// TIA Portal project "MB TCP S7-1200 - HMI ET6600" (V19)

(* hardware
DEVICE "S7-1200 station_1"  S7-1200 Station
   slot 0: "Rack_0"  S7-1200 Rack  Rack  V1.0
   slot 1: "PLC_1"  CPU 1215C DC/DC/DC  6ES7 215-1AG40-0XB0  V4.5
*)

// ===== PLC "PLC_1"  CPU 1215C DC/DC/DC =====

VAR_GLOBAL   // PLC tag table "Default tag table"
   "Encendido" AT %M0.0 : Bool;
   "ManAuto" AT %M0.1 : Bool;
   "System_Byte" AT %MB1 : Byte;
   "FirstScan" AT %M1.0 : Bool;
   "DiagStatusUpdate" AT %M1.1 : Bool;
   "AlwaysTRUE" AT %M1.2 : Bool;
   "AlwaysFALSE" AT %M1.3 : Bool;
END_VAR

DATA_BLOCK "DB_AproxTemp"   // DB1
{ S7_Optimized_Access := 'TRUE' }
VERSION : 0.1
// stored: InstanceOfName FB_Aprox
"FB_Aprox"
BEGIN
END_DATA_BLOCK

DATA_BLOCK "DB_HMIET"   // DB2
{ S7_Optimized_Access := 'FALSE' }
VERSION : 0.1
   VAR
      TEMPERATURA_SP : Real := 22.0;
      HUMEDAD_SP : Real := 60.0;
      PRESION_SP : Real := 1015.0;
      VENT_VEL_OUT : Real := 799.0;
      BOMBA_VEL_OUT : Real := 1434.0;
      TEMPERATURA_HMI : Int;
      HUMEDAD_HMI : Int;
      PRESION_HMI : Int;
      ENFRIAMIENTO_HMI : Bool;
      CALEFACCION_HMI : Bool;
      DESHUM_HMI : Bool;
      AutoMan : Bool;
      CAUDAL_BS : Int;
      MrgPre : Real;
   END_VAR
BEGIN
END_DATA_BLOCK

DATA_BLOCK "DB_AproxHum"   // DB3
{ S7_Optimized_Access := 'TRUE' }
VERSION : 0.1
// stored: InstanceOfName FB_Aprox
"FB_Aprox"
BEGIN
END_DATA_BLOCK

DATA_BLOCK "DB_AproxPre"   // DB4
{ S7_Optimized_Access := 'TRUE' }
VERSION : 0.1
// stored: InstanceOfName FB_Aprox
"FB_Aprox"
BEGIN
END_DATA_BLOCK

DATA_BLOCK "DB_SimTemp"   // DB5
{ S7_Optimized_Access := 'TRUE' }
VERSION : 0.1
// stored: InstanceOfName FB_Simulacion
"FB_Simulacion"
BEGIN
END_DATA_BLOCK

DATA_BLOCK "DB_SimPre"   // DB6
{ S7_Optimized_Access := 'TRUE' }
VERSION : 0.1
// stored: InstanceOfName FB_Simulacion
"FB_Simulacion"
BEGIN
END_DATA_BLOCK

DATA_BLOCK "DB_HMIOUT"   // DB7
{ S7_Optimized_Access := 'FALSE' }
VERSION : 0.1
   VAR
      PRESION_OUT : Real;
      HUMEDAD_OUT : Real;
      TEMPERATURA_OUT : Real;
      TENSION_OUT : Real;
      CORRIENTE_OUT : Real;
      VELOCIDAD_OUT : Real;
      PPM_PRC : Int;
      PPM_OUT : Int;
      ALARMA_BS : Bool;
   END_VAR
BEGIN
END_DATA_BLOCK

DATA_BLOCK "DB_OsciladorTension"   // DB8
{ S7_Optimized_Access := 'TRUE' }
VERSION : 0.1
// stored: InstanceOfName FB_Oscilador
"FB_Oscilador"
BEGIN
END_DATA_BLOCK

DATA_BLOCK "DB_OsciladorCorriente"   // DB9
{ S7_Optimized_Access := 'TRUE' }
VERSION : 0.1
// stored: InstanceOfName FB_Oscilador
"FB_Oscilador"
BEGIN
END_DATA_BLOCK

DATA_BLOCK "DB_OsciladorVel"   // DB10
{ S7_Optimized_Access := 'TRUE' }
VERSION : 0.1
// stored: InstanceOfName FB_Oscilador
"FB_Oscilador"
BEGIN
END_DATA_BLOCK

DATA_BLOCK "DB_CaliAire"   // DB11
{ S7_Optimized_Access := 'TRUE' }
VERSION : 0.1
// stored: InstanceOfName FB_CaliAire
"FB_CaliAire"
BEGIN
END_DATA_BLOCK

DATA_BLOCK "DB_SimHum"   // DB12
{ S7_Optimized_Access := 'TRUE' }
VERSION : 0.1
// stored: InstanceOfName FB_Simulacion
"FB_Simulacion"
BEGIN
END_DATA_BLOCK

// folder: System blocks/Program resources

DATA_BLOCK "Timer_VelBombaVent"   // DB13
{ S7_Optimized_Access := 'TRUE' }
AUTHOR : Simatic
FAMILY : IEC
NAME : IEC_TMR
VERSION : 1.0
// stored: InstanceOfName IEC_TIMER
"IEC_TIMER"
BEGIN
END_DATA_BLOCK

// folder: (top level)

FUNCTION_BLOCK "FB_Oscilador"   // FB1, LAD
{ S7_Optimized_Access := 'TRUE' }
VERSION : 0.1
   VAR_INPUT
      SP : Real;
      MS : Real;
      MI : Real;
      Tiempo : Time;
      Enc : Bool;
   END_VAR
   VAR_OUTPUT
      PV : Real;
   END_VAR
   VAR
      Timer_MS : TON_TIME;
      Reset_TMS : Bool;
      Timer_ResetMS : TON_TIME;
      Intermedio : Bool;
      Reset_TMI : Bool;
      Timer_MI : TON_TIME;
      Timer_ResetMI : TON_TIME;
   END_VAR
BEGIN

REGION Network 1
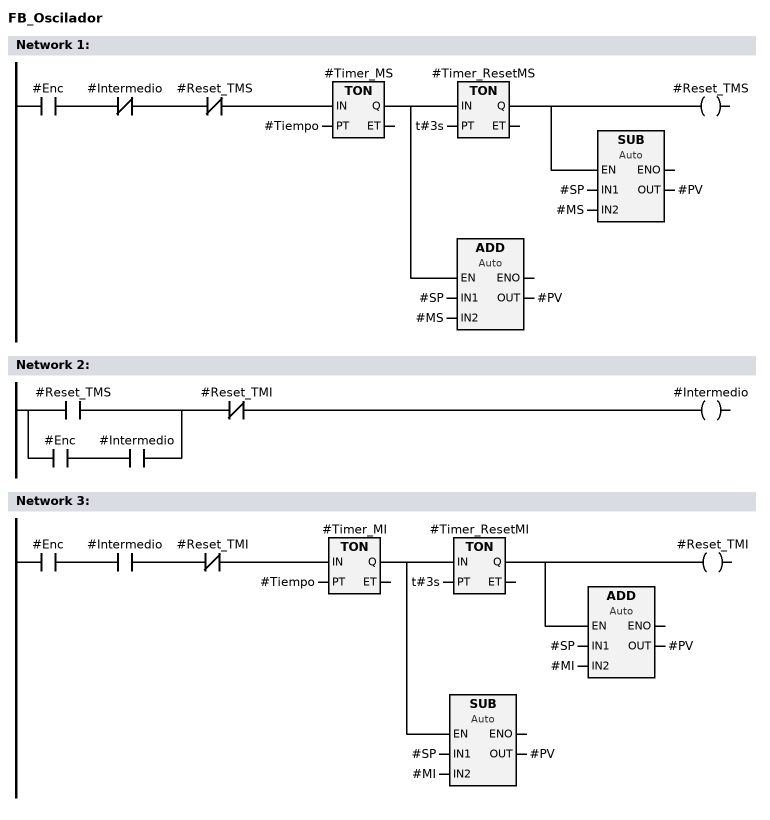
   #Timer_MS(IN := #Enc AND NOT #Intermedio AND NOT #Reset_TMS, PT := #Tiempo);   // TON
   #Timer_ResetMS(IN := #Timer_MS.Q, PT := t#3s);   // TON
   #Reset_TMS := #Timer_ResetMS.Q;
   IF #Timer_ResetMS.Q THEN #PV := #SP - #MS; END_IF;
   IF #Timer_MS.Q THEN #PV := #SP + #MS; END_IF;
END_REGION

REGION Network 2
   RUNG wire#powerrail
      Contact( #Reset_TMS )
      wire#w1
      I_Contact( #Reset_TMI )
      Coil( #Intermedio )
   END_RUNG
   RUNG wire#powerrail
      Contact( #Enc )
      Contact( #Intermedio )
   END_RUNG wire#w1
   // the same network as SCL:
   #Intermedio := (#Reset_TMS OR (#Enc AND #Intermedio)) AND NOT #Reset_TMI;
END_REGION

REGION Network 3
   #Timer_MI(IN := #Enc AND #Intermedio AND NOT #Reset_TMI, PT := #Tiempo);   // TON
   #Timer_ResetMI(IN := #Timer_MI.Q, PT := t#3s);   // TON
   #Reset_TMI := #Timer_ResetMI.Q;
   IF #Timer_ResetMI.Q THEN #PV := #SP + #MI; END_IF;
   IF #Timer_MI.Q THEN #PV := #SP - #MI; END_IF;
END_REGION
END_FUNCTION_BLOCK

FUNCTION_BLOCK "FB_Simulacion"   // FB2, LAD
{ S7_Optimized_Access := 'TRUE' }
VERSION : 0.1
   VAR_INPUT
      Enc : Bool;
      Mrg : Real;
   END_VAR
   VAR_OUTPUT
      PV : Real;
      Ctrl : Int;
      Sim : Bool;
   END_VAR
   VAR
      Aux : Array[0..7] of Bool;
      MarcaEnc : Bool;
      TimerSuma : TON_TIME;
      TimerEnclavSuma : TON_TIME;
      TimerDelay : TON_TIME;
      TimerEnclavResta : TON_TIME;
   END_VAR
   VAR_TEMP   // added for the SCL form of the ladder/FBD networks
      _w1 : Bool;
   END_VAR
BEGIN

REGION Network 1
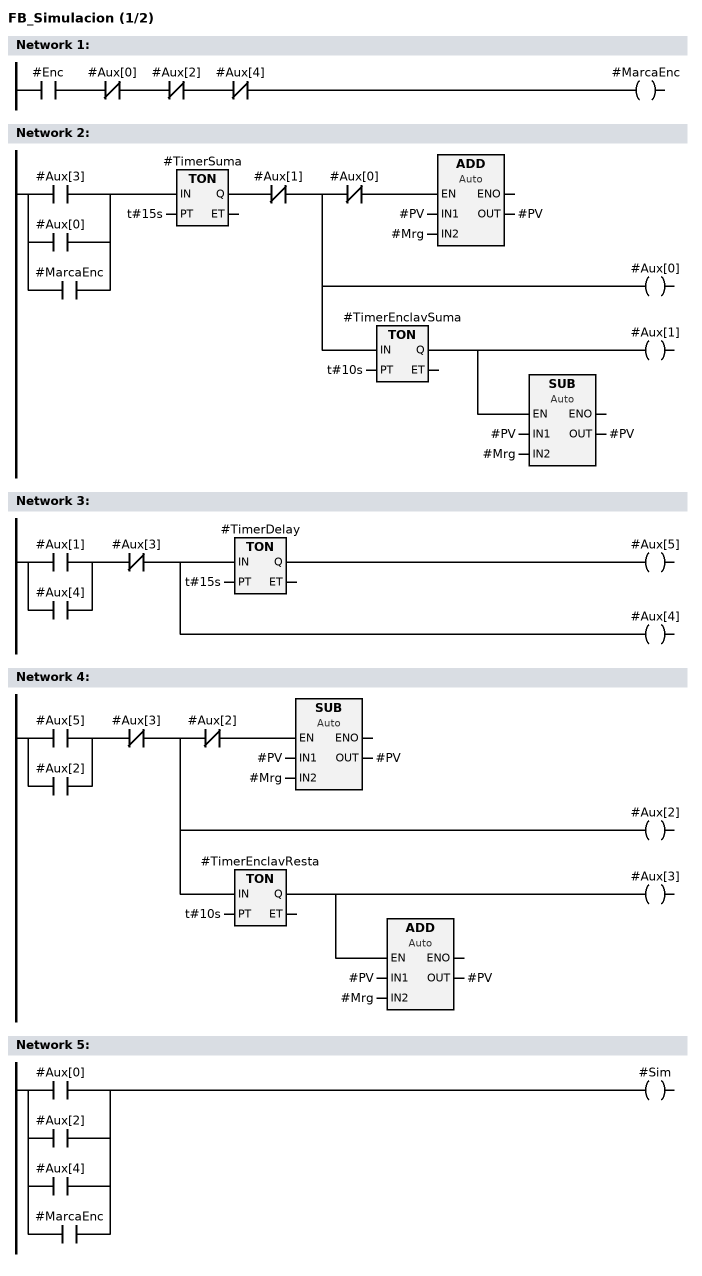
   RUNG wire#powerrail
      Contact( #Enc )
      I_Contact( #Aux[0] )
      I_Contact( #Aux[2] )
      I_Contact( #Aux[4] )
      Coil( #MarcaEnc )
   END_RUNG
   // the same network as SCL:
   #MarcaEnc := #Enc AND NOT #Aux[0] AND NOT #Aux[2] AND NOT #Aux[4];
END_REGION

REGION Network 2
   #TimerSuma(IN := #Aux[3] OR #Aux[0] OR #MarcaEnc, PT := t#15s);   // TON
   #_w1 := #TimerSuma.Q AND NOT #Aux[1];
   IF #_w1 AND NOT #Aux[0] THEN #PV := #PV + #Mrg; END_IF;
   #Aux[0] := #_w1;
   #TimerEnclavSuma(IN := #_w1, PT := t#10s);   // TON
   #Aux[1] := #TimerEnclavSuma.Q;
   IF #TimerEnclavSuma.Q THEN #PV := #PV - #Mrg; END_IF;
END_REGION

REGION Network 3
   #_w1 := (#Aux[1] OR #Aux[4]) AND NOT #Aux[3];
   #TimerDelay(IN := #_w1, PT := t#15s);   // TON
   #Aux[5] := #TimerDelay.Q;
   #Aux[4] := #_w1;
END_REGION

REGION Network 4
   #_w1 := (#Aux[5] OR #Aux[2]) AND NOT #Aux[3];
   IF #_w1 AND NOT #Aux[2] THEN #PV := #PV - #Mrg; END_IF;
   #Aux[2] := #_w1;
   #TimerEnclavResta(IN := #_w1, PT := t#10s);   // TON
   #Aux[3] := #TimerEnclavResta.Q;
   IF #TimerEnclavResta.Q THEN #PV := #PV + #Mrg; END_IF;
END_REGION

REGION Network 5
   RUNG wire#powerrail
      Contact( #Aux[0] )
      wire#w1
      Coil( #Sim )
   END_RUNG
   RUNG wire#powerrail
      Contact( #Aux[2] )
   END_RUNG wire#w1
   RUNG wire#powerrail
      Contact( #Aux[4] )
   END_RUNG wire#w1
   RUNG wire#powerrail
      Contact( #MarcaEnc )
   END_RUNG wire#w1
   // the same network as SCL:
   #Sim := #Aux[0] OR #Aux[2] OR #Aux[4] OR #MarcaEnc;
END_REGION

REGION Network 6
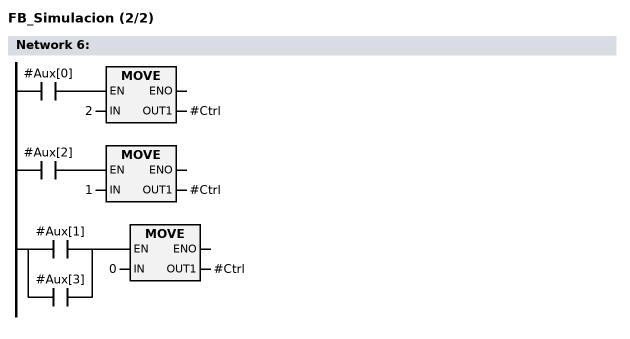
   RUNG wire#powerrail
      Contact( #Aux[0] )
      Move(in := 2, out1 => #Ctrl)
   END_RUNG
   RUNG wire#powerrail
      Contact( #Aux[2] )
      Move(in := 1, out1 => #Ctrl)
   END_RUNG
   RUNG wire#powerrail
      Contact( #Aux[1] )
      wire#w1
      Move(in := 0, out1 => #Ctrl)
   END_RUNG
   RUNG wire#powerrail
      Contact( #Aux[3] )
   END_RUNG wire#w1
   // the same network as SCL:
   IF #Aux[0] THEN #Ctrl := 2; END_IF;
   IF #Aux[2] THEN #Ctrl := 1; END_IF;
   IF #Aux[1] OR #Aux[3] THEN #Ctrl := 0; END_IF;
END_REGION
END_FUNCTION_BLOCK

FUNCTION_BLOCK "FB_CaliAire"   // FB3, LAD
{ S7_Optimized_Access := 'TRUE' }
VERSION : 0.1
   VAR_INPUT
      Caudal : Int;
      Lim : Int;
   END_VAR
   VAR_OUTPUT
      PPM : Int;
      PPMEsc : Int;
      Alarma : Bool;
   END_VAR
   VAR
      UltCaudal : Int := 100;
      TempOn : Bool;
      Timer_CaliAire : TON_TIME;
      TempPPM : Real;
   END_VAR
BEGIN

REGION Network 1
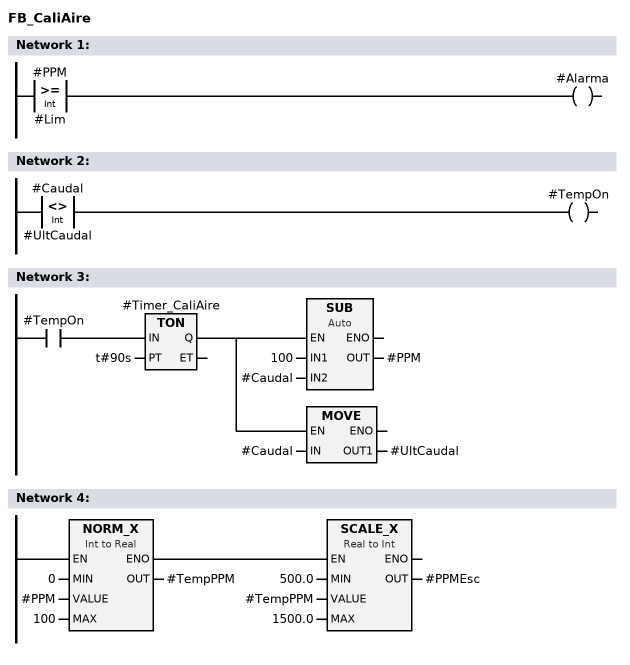
   RUNG wire#powerrail
      { S7_Templates := "SrcType := Int" } GE_Contact(in1 := #PPM, in2 := #Lim)
      Coil( #Alarma )
   END_RUNG
   // the same network as SCL:
   #Alarma := #PPM >= #Lim;
END_REGION

REGION Network 2
   RUNG wire#powerrail
      { S7_Templates := "SrcType := Int" } NE_Contact(in1 := #Caudal, in2 := #UltCaudal)
      Coil( #TempOn )
   END_RUNG
   // the same network as SCL:
   #TempOn := #Caudal <> #UltCaudal;
END_REGION

REGION Network 3
   #Timer_CaliAire(IN := #TempOn, PT := t#90s);   // TON
   IF #Timer_CaliAire.Q THEN
       #PPM := 100 - #Caudal;
       #UltCaudal := #Caudal;
   END_IF;
END_REGION

REGION Network 4
   RUNG wire#powerrail
      { S7_Templates := "[SrcType := Int, DestType := Real]" } Normalize(min := 0, value := #PPM, max := 100, out => #TempPPM)
      { S7_Templates := "[SrcType := Real, DestType := Int]" } Scale(min := 500.0, value := #TempPPM, max := 1500.0, out => #PPMEsc)
   END_RUNG
   // the same network as SCL:
   #TempPPM := NORM_X(MIN := 0, VALUE := #PPM, MAX := 100);
   #PPMEsc := SCALE_X(MIN := 500.0, VALUE := #TempPPM, MAX := 1500.0);
END_REGION
END_FUNCTION_BLOCK

FUNCTION_BLOCK "FB_Aprox"   // FB4, LAD
{ S7_Optimized_Access := 'TRUE' }
VERSION : 0.1
   VAR_INPUT
      Enc : Bool;
      SP : Real;
      Mrg : Real;
   END_VAR
   VAR_OUTPUT
      PV : Real;
      Ctrl : Int;
   END_VAR
   VAR
      Aux : Array[0..7] of Bool;
      TimerAprox : TON_TIME;
   END_VAR
BEGIN

REGION Network 1
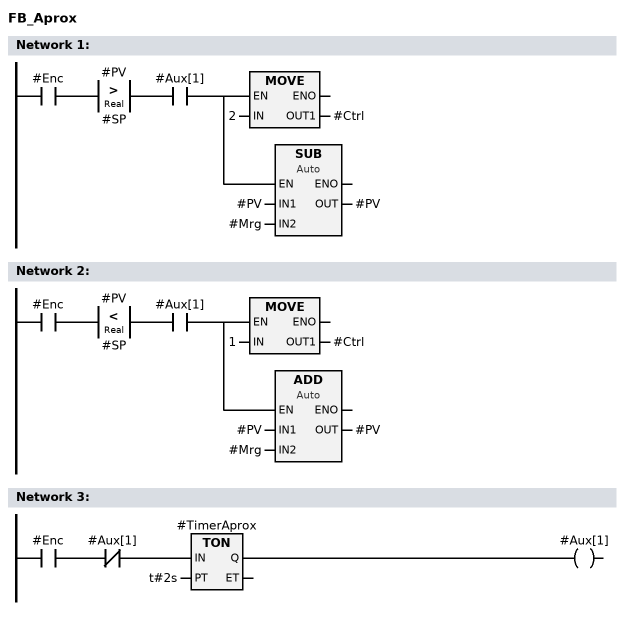
   RUNG wire#powerrail
      Contact( #Enc )
      { S7_Templates := "SrcType := Real" } GT_Contact(in1 := #PV, in2 := #SP)
      Contact( #Aux[1] )
      wire#w1
      Move(in := 2, out1 => #Ctrl)
   END_RUNG
   RUNG wire#w1
      Sub(in1 := #PV, in2 := #Mrg, out => #PV)
   END_RUNG
   // the same network as SCL:
   IF #Enc AND (#PV > #SP) AND #Aux[1] THEN
       #Ctrl := 2;
       #PV := #PV - #Mrg;
   END_IF;
END_REGION

REGION Network 2
   RUNG wire#powerrail
      Contact( #Enc )
      { S7_Templates := "SrcType := Real" } LT_Contact(in1 := #PV, in2 := #SP)
      Contact( #Aux[1] )
      wire#w1
      Move(in := 1, out1 => #Ctrl)
   END_RUNG
   RUNG wire#w1
      Add(in1 := #PV, in2 := #Mrg, out => #PV)
   END_RUNG
   // the same network as SCL:
   IF #Enc AND (#PV < #SP) AND #Aux[1] THEN
       #Ctrl := 1;
       #PV := #PV + #Mrg;
   END_IF;
END_REGION

REGION Network 3
   #TimerAprox(IN := #Enc AND NOT #Aux[1], PT := t#2s);   // TON
   #Aux[1] := #TimerAprox.Q;
END_REGION
END_FUNCTION_BLOCK

FUNCTION_BLOCK "Modbus_TCP"   // FB5, LAD
{ S7_Optimized_Access := 'TRUE' }
VERSION : 0.1
BEGIN
END_FUNCTION_BLOCK

FUNCTION "FC_ConversionEscalado" : Void   // FC1, LAD
{ S7_Optimized_Access := 'TRUE' }
VERSION : 0.1
   VAR_INPUT
      EntradaInt : Int;
      MinNorm : Int;
      MaxNorm : Int;
      MinReal : Real;
      MaxReal : Real;
   END_VAR
   VAR_OUTPUT
      SalidaReal : Real;
   END_VAR
   VAR_TEMP
      IntReal : Real;
      RealNorm : Real;
   END_VAR
BEGIN

REGION Network 1
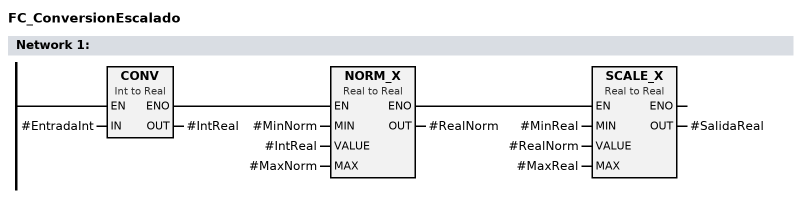
   RUNG wire#powerrail
      { S7_Templates := "[SrcType := Int, DestType := Real]" } Convert(in := #EntradaInt, out => #IntReal)
      { S7_Templates := "[SrcType := Real, DestType := Real]" } Normalize(min := #MinNorm, value := #IntReal, max := #MaxNorm, out => #RealNorm)
      { S7_Templates := "[SrcType := Real, DestType := Real]" } Scale(min := #MinReal, value := #RealNorm, max := #MaxReal, out => #SalidaReal)
   END_RUNG
   // the same network as SCL:
   #IntReal := INT_TO_REAL(#EntradaInt);
   #RealNorm := NORM_X(MIN := #MinNorm, VALUE := #IntReal, MAX := #MaxNorm);
   #SalidaReal := SCALE_X(MIN := #MinReal, VALUE := #RealNorm, MAX := #MaxReal);
END_REGION
END_FUNCTION

ORGANIZATION_BLOCK "Main"   // OB1, LAD, ProgramCycle
TITLE = "Main Program Sweep (Cycle)"
{ S7_Optimized_Access := 'TRUE' }
VERSION : 0.1
   VAR_INPUT
      Initial_Call : Bool;   // Initial call of this OB
      Remanence : Bool;   // =True, if remanent data are available
   END_VAR
   VAR_TEMP
      SPTEMP_ESC : Real;
      SPHUM_ESC : Real;
      SPPRE_ESC : Real;
   END_VAR
BEGIN

REGION Network 1
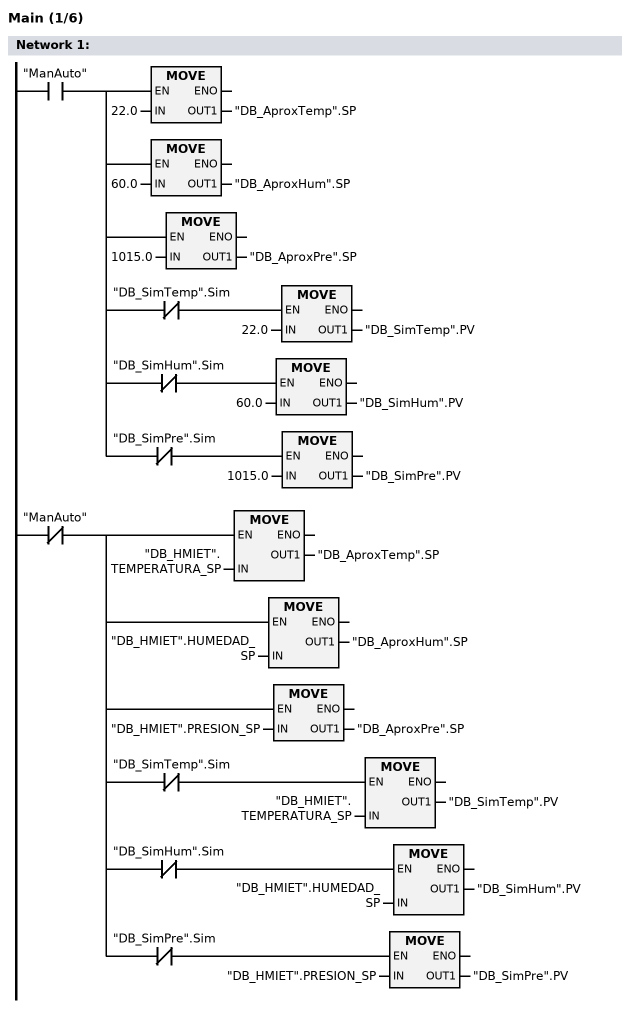
   RUNG wire#powerrail
      Contact( "ManAuto" )
      wire#w1
      Move(in := 22.0, out1 => "DB_AproxTemp".SP)
   END_RUNG
   RUNG wire#w1
      Move(in := 60.0, out1 => "DB_AproxHum".SP)
   END_RUNG
   RUNG wire#w1
      Move(in := 1015.0, out1 => "DB_AproxPre".SP)
   END_RUNG
   RUNG wire#w1
      I_Contact( "DB_SimTemp".Sim )
      Move(in := 22.0, out1 => "DB_SimTemp".PV)
   END_RUNG
   RUNG wire#w1
      I_Contact( "DB_SimHum".Sim )
      Move(in := 60.0, out1 => "DB_SimHum".PV)
   END_RUNG
   RUNG wire#w1
      I_Contact( "DB_SimPre".Sim )
      Move(in := 1015.0, out1 => "DB_SimPre".PV)
   END_RUNG
   RUNG wire#powerrail
      I_Contact( "ManAuto" )
      wire#w2
      Move(in := "DB_HMIET".TEMPERATURA_SP, out1 => "DB_AproxTemp".SP)
   END_RUNG
   RUNG wire#w2
      Move(in := "DB_HMIET".HUMEDAD_SP, out1 => "DB_AproxHum".SP)
   END_RUNG
   RUNG wire#w2
      Move(in := "DB_HMIET".PRESION_SP, out1 => "DB_AproxPre".SP)
   END_RUNG
   RUNG wire#w2
      I_Contact( "DB_SimTemp".Sim )
      Move(in := "DB_HMIET".TEMPERATURA_SP, out1 => "DB_SimTemp".PV)
   END_RUNG
   RUNG wire#w2
      I_Contact( "DB_SimHum".Sim )
      Move(in := "DB_HMIET".HUMEDAD_SP, out1 => "DB_SimHum".PV)
   END_RUNG
   RUNG wire#w2
      I_Contact( "DB_SimPre".Sim )
      Move(in := "DB_HMIET".PRESION_SP, out1 => "DB_SimPre".PV)
   END_RUNG
   // the same network as SCL:
   IF "ManAuto" THEN
       "DB_AproxTemp".SP := 22.0;
       "DB_AproxHum".SP := 60.0;
       "DB_AproxPre".SP := 1015.0;
   END_IF;
   IF "ManAuto" AND NOT "DB_SimTemp".Sim THEN "DB_SimTemp".PV := 22.0; END_IF;
   IF "ManAuto" AND NOT "DB_SimHum".Sim THEN "DB_SimHum".PV := 60.0; END_IF;
   IF "ManAuto" AND NOT "DB_SimPre".Sim THEN "DB_SimPre".PV := 1015.0; END_IF;
   IF NOT "ManAuto" THEN
       "DB_AproxTemp".SP := "DB_HMIET".TEMPERATURA_SP;
       "DB_AproxHum".SP := "DB_HMIET".HUMEDAD_SP;
       "DB_AproxPre".SP := "DB_HMIET".PRESION_SP;
   END_IF;
   IF NOT "ManAuto" AND NOT "DB_SimTemp".Sim THEN "DB_SimTemp".PV := "DB_HMIET".TEMPERATURA_SP; END_IF;
   IF NOT "ManAuto" AND NOT "DB_SimHum".Sim THEN "DB_SimHum".PV := "DB_HMIET".HUMEDAD_SP; END_IF;
   IF NOT "ManAuto" AND NOT "DB_SimPre".Sim THEN "DB_SimPre".PV := "DB_HMIET".PRESION_SP; END_IF;
END_REGION

REGION Network 2
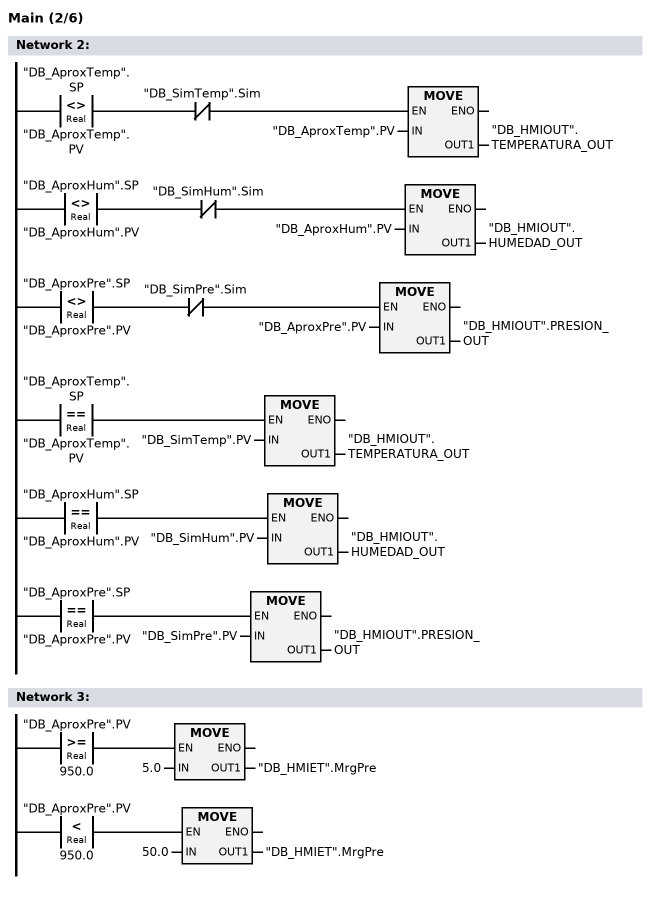
   RUNG wire#powerrail
      { S7_Templates := "SrcType := Real" } NE_Contact(in1 := "DB_AproxTemp".SP, in2 := "DB_AproxTemp".PV)
      I_Contact( "DB_SimTemp".Sim )
      Move(in := "DB_AproxTemp".PV, out1 => "DB_HMIOUT".TEMPERATURA_OUT)
   END_RUNG
   RUNG wire#powerrail
      { S7_Templates := "SrcType := Real" } NE_Contact(in1 := "DB_AproxHum".SP, in2 := "DB_AproxHum".PV)
      I_Contact( "DB_SimHum".Sim )
      Move(in := "DB_AproxHum".PV, out1 => "DB_HMIOUT".HUMEDAD_OUT)
   END_RUNG
   RUNG wire#powerrail
      { S7_Templates := "SrcType := Real" } NE_Contact(in1 := "DB_AproxPre".SP, in2 := "DB_AproxPre".PV)
      I_Contact( "DB_SimPre".Sim )
      Move(in := "DB_AproxPre".PV, out1 => "DB_HMIOUT".PRESION_OUT)
   END_RUNG
   RUNG wire#powerrail
      { S7_Templates := "SrcType := Real" } EQ_Contact(in1 := "DB_AproxTemp".SP, in2 := "DB_AproxTemp".PV)
      Move(in := "DB_SimTemp".PV, out1 => "DB_HMIOUT".TEMPERATURA_OUT)
   END_RUNG
   RUNG wire#powerrail
      { S7_Templates := "SrcType := Real" } EQ_Contact(in1 := "DB_AproxHum".SP, in2 := "DB_AproxHum".PV)
      Move(in := "DB_SimHum".PV, out1 => "DB_HMIOUT".HUMEDAD_OUT)
   END_RUNG
   RUNG wire#powerrail
      { S7_Templates := "SrcType := Real" } EQ_Contact(in1 := "DB_AproxPre".SP, in2 := "DB_AproxPre".PV)
      Move(in := "DB_SimPre".PV, out1 => "DB_HMIOUT".PRESION_OUT)
   END_RUNG
   // the same network as SCL:
   IF ("DB_AproxTemp".SP <> "DB_AproxTemp".PV) AND NOT "DB_SimTemp".Sim THEN
       "DB_HMIOUT".TEMPERATURA_OUT := "DB_AproxTemp".PV;
   END_IF;
   IF ("DB_AproxHum".SP <> "DB_AproxHum".PV) AND NOT "DB_SimHum".Sim THEN
       "DB_HMIOUT".HUMEDAD_OUT := "DB_AproxHum".PV;
   END_IF;
   IF ("DB_AproxPre".SP <> "DB_AproxPre".PV) AND NOT "DB_SimPre".Sim THEN
       "DB_HMIOUT".PRESION_OUT := "DB_AproxPre".PV;
   END_IF;
   IF "DB_AproxTemp".SP = "DB_AproxTemp".PV THEN "DB_HMIOUT".TEMPERATURA_OUT := "DB_SimTemp".PV; END_IF;
   IF "DB_AproxHum".SP = "DB_AproxHum".PV THEN "DB_HMIOUT".HUMEDAD_OUT := "DB_SimHum".PV; END_IF;
   IF "DB_AproxPre".SP = "DB_AproxPre".PV THEN "DB_HMIOUT".PRESION_OUT := "DB_SimPre".PV; END_IF;
END_REGION

REGION Network 3
   RUNG wire#powerrail
      { S7_Templates := "SrcType := Real" } GE_Contact(in1 := "DB_AproxPre".PV, in2 := 950.0)
      Move(in := 5.0, out1 => "DB_HMIET".MrgPre)
   END_RUNG
   RUNG wire#powerrail
      { S7_Templates := "SrcType := Real" } LT_Contact(in1 := "DB_AproxPre".PV, in2 := 950.0)
      Move(in := 50.0, out1 => "DB_HMIET".MrgPre)
   END_RUNG
   // the same network as SCL:
   IF "DB_AproxPre".PV >= 950.0 THEN "DB_HMIET".MrgPre := 5.0; END_IF;
   IF "DB_AproxPre".PV < 950.0 THEN "DB_HMIET".MrgPre := 50.0; END_IF;
END_REGION

REGION Network 4
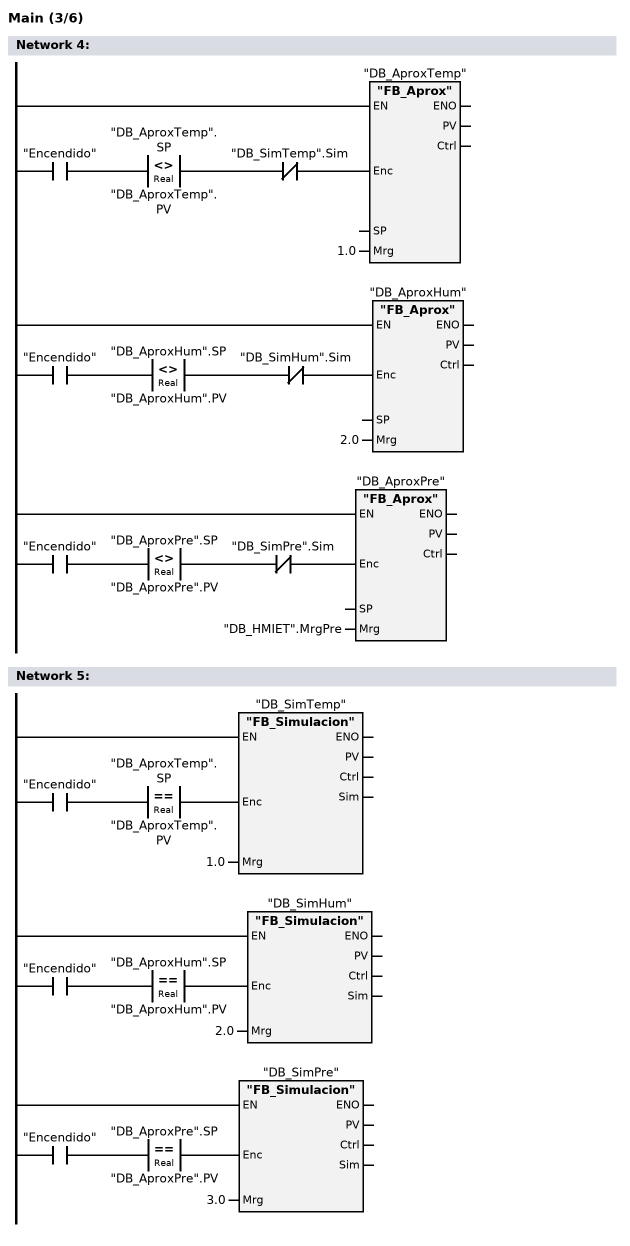
   RUNG wire#powerrail
      "DB_AproxTemp"(Enc := wire#w1, SP :=, Mrg := 1.0, PV =>, Ctrl =>)
   END_RUNG
   RUNG wire#powerrail
      Contact( "Encendido" )
      { S7_Templates := "SrcType := Real" } NE_Contact(in1 := "DB_AproxTemp".SP, in2 := "DB_AproxTemp".PV)
      I_Contact( "DB_SimTemp".Sim )
   END_RUNG wire#w1
   RUNG wire#powerrail
      "DB_AproxHum"(Enc := wire#w2, SP :=, Mrg := 2.0, PV =>, Ctrl =>)
   END_RUNG
   RUNG wire#powerrail
      Contact( "Encendido" )
      { S7_Templates := "SrcType := Real" } NE_Contact(in1 := "DB_AproxHum".SP, in2 := "DB_AproxHum".PV)
      I_Contact( "DB_SimHum".Sim )
   END_RUNG wire#w2
   RUNG wire#powerrail
      "DB_AproxPre"(Enc := wire#w3, SP :=, Mrg := "DB_HMIET".MrgPre, PV =>, Ctrl =>)
   END_RUNG
   RUNG wire#powerrail
      Contact( "Encendido" )
      { S7_Templates := "SrcType := Real" } NE_Contact(in1 := "DB_AproxPre".SP, in2 := "DB_AproxPre".PV)
      I_Contact( "DB_SimPre".Sim )
   END_RUNG wire#w3
   // the same network as SCL:
   "DB_AproxTemp"(Enc := "Encendido" AND ("DB_AproxTemp".SP <> "DB_AproxTemp".PV) AND NOT "DB_SimTemp".Sim,   // "FB_Aprox"
                  Mrg := 1.0);
   "DB_AproxHum"(Enc := "Encendido" AND ("DB_AproxHum".SP <> "DB_AproxHum".PV) AND NOT "DB_SimHum".Sim,   // "FB_Aprox"
                 Mrg := 2.0);
   "DB_AproxPre"(Enc := "Encendido" AND ("DB_AproxPre".SP <> "DB_AproxPre".PV) AND NOT "DB_SimPre".Sim,   // "FB_Aprox"
                 Mrg := "DB_HMIET".MrgPre);
END_REGION

REGION Network 5
   RUNG wire#powerrail
      "DB_SimTemp"(Enc := wire#w1, Mrg := 1.0, PV =>, Ctrl =>, Sim =>)
   END_RUNG
   RUNG wire#powerrail
      Contact( "Encendido" )
      { S7_Templates := "SrcType := Real" } EQ_Contact(in1 := "DB_AproxTemp".SP, in2 := "DB_AproxTemp".PV)
   END_RUNG wire#w1
   RUNG wire#powerrail
      "DB_SimHum"(Enc := wire#w2, Mrg := 2.0, PV =>, Ctrl =>, Sim =>)
   END_RUNG
   RUNG wire#powerrail
      Contact( "Encendido" )
      { S7_Templates := "SrcType := Real" } EQ_Contact(in1 := "DB_AproxHum".SP, in2 := "DB_AproxHum".PV)
   END_RUNG wire#w2
   RUNG wire#powerrail
      "DB_SimPre"(Enc := wire#w3, Mrg := 3.0, PV =>, Ctrl =>, Sim =>)
   END_RUNG
   RUNG wire#powerrail
      Contact( "Encendido" )
      { S7_Templates := "SrcType := Real" } EQ_Contact(in1 := "DB_AproxPre".SP, in2 := "DB_AproxPre".PV)
   END_RUNG wire#w3
   // the same network as SCL:
   "DB_SimTemp"(Enc := "Encendido" AND ("DB_AproxTemp".SP = "DB_AproxTemp".PV), Mrg := 1.0);   // "FB_Simulacion"
   "DB_SimHum"(Enc := "Encendido" AND ("DB_AproxHum".SP = "DB_AproxHum".PV), Mrg := 2.0);   // "FB_Simulacion"
   "DB_SimPre"(Enc := "Encendido" AND ("DB_AproxPre".SP = "DB_AproxPre".PV), Mrg := 3.0);   // "FB_Simulacion"
END_REGION

REGION Network 6
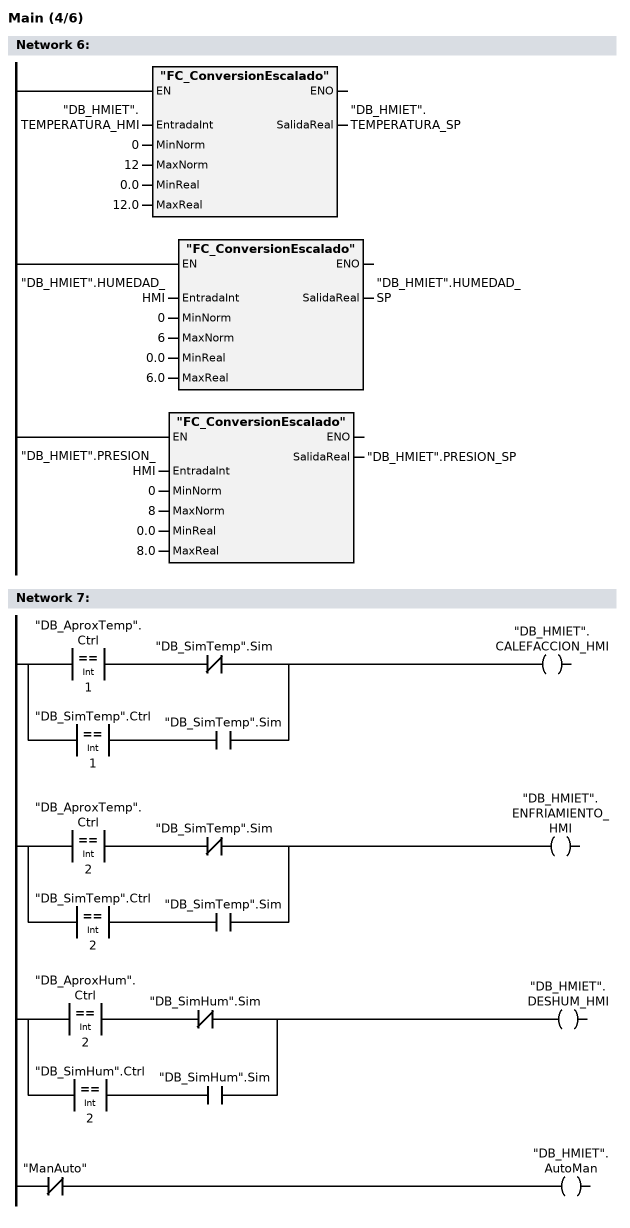
   RUNG wire#powerrail
      "FC_ConversionEscalado"(EntradaInt := "DB_HMIET".TEMPERATURA_HMI, MinNorm := 0, MaxNorm := 12, MinReal := 0.0, MaxReal := 12.0, SalidaReal => "DB_HMIET".TEMPERATURA_SP)
   END_RUNG
   RUNG wire#powerrail
      "FC_ConversionEscalado"(EntradaInt := "DB_HMIET".HUMEDAD_HMI, MinNorm := 0, MaxNorm := 6, MinReal := 0.0, MaxReal := 6.0, SalidaReal => "DB_HMIET".HUMEDAD_SP)
   END_RUNG
   RUNG wire#powerrail
      "FC_ConversionEscalado"(EntradaInt := "DB_HMIET".PRESION_HMI, MinNorm := 0, MaxNorm := 8, MinReal := 0.0, MaxReal := 8.0, SalidaReal => "DB_HMIET".PRESION_SP)
   END_RUNG
   // the same network as SCL:
   "FC_ConversionEscalado"(EntradaInt := "DB_HMIET".TEMPERATURA_HMI,
                           MinNorm := 0,
                           MaxNorm := 12,
                           MinReal := 0.0,
                           MaxReal := 12.0,
                           SalidaReal => "DB_HMIET".TEMPERATURA_SP);
   "FC_ConversionEscalado"(EntradaInt := "DB_HMIET".HUMEDAD_HMI,
                           MinNorm := 0,
                           MaxNorm := 6,
                           MinReal := 0.0,
                           MaxReal := 6.0,
                           SalidaReal => "DB_HMIET".HUMEDAD_SP);
   "FC_ConversionEscalado"(EntradaInt := "DB_HMIET".PRESION_HMI,
                           MinNorm := 0,
                           MaxNorm := 8,
                           MinReal := 0.0,
                           MaxReal := 8.0,
                           SalidaReal => "DB_HMIET".PRESION_SP);
END_REGION

REGION Network 7
   RUNG wire#powerrail
      { S7_Templates := "SrcType := Int" } EQ_Contact(in1 := "DB_AproxTemp".Ctrl, in2 := 1)
      I_Contact( "DB_SimTemp".Sim )
      wire#w1
      Coil( "DB_HMIET".CALEFACCION_HMI )
   END_RUNG
   RUNG wire#powerrail
      { S7_Templates := "SrcType := Int" } EQ_Contact(in1 := "DB_SimTemp".Ctrl, in2 := 1)
      Contact( "DB_SimTemp".Sim )
   END_RUNG wire#w1
   RUNG wire#powerrail
      { S7_Templates := "SrcType := Int" } EQ_Contact(in1 := "DB_AproxTemp".Ctrl, in2 := 2)
      I_Contact( "DB_SimTemp".Sim )
      wire#w2
      Coil( "DB_HMIET".ENFRIAMIENTO_HMI )
   END_RUNG
   RUNG wire#powerrail
      { S7_Templates := "SrcType := Int" } EQ_Contact(in1 := "DB_SimTemp".Ctrl, in2 := 2)
      Contact( "DB_SimTemp".Sim )
   END_RUNG wire#w2
   RUNG wire#powerrail
      { S7_Templates := "SrcType := Int" } EQ_Contact(in1 := "DB_AproxHum".Ctrl, in2 := 2)
      I_Contact( "DB_SimHum".Sim )
      wire#w3
      Coil( "DB_HMIET".DESHUM_HMI )
   END_RUNG
   RUNG wire#powerrail
      { S7_Templates := "SrcType := Int" } EQ_Contact(in1 := "DB_SimHum".Ctrl, in2 := 2)
      Contact( "DB_SimHum".Sim )
   END_RUNG wire#w3
   RUNG wire#powerrail
      I_Contact( "ManAuto" )
      Coil( "DB_HMIET".AutoMan )
   END_RUNG
   // the same network as SCL:
   "DB_HMIET".CALEFACCION_HMI := (("DB_AproxTemp".Ctrl = 1) AND NOT "DB_SimTemp".Sim) OR (("DB_SimTemp".Ctrl = 1) AND "DB_SimTemp".Sim);
   "DB_HMIET".ENFRIAMIENTO_HMI := (("DB_AproxTemp".Ctrl = 2) AND NOT "DB_SimTemp".Sim) OR (("DB_SimTemp".Ctrl = 2) AND "DB_SimTemp".Sim);
   "DB_HMIET".DESHUM_HMI := (("DB_AproxHum".Ctrl = 2) AND NOT "DB_SimHum".Sim) OR (("DB_SimHum".Ctrl = 2) AND "DB_SimHum".Sim);
   "DB_HMIET".AutoMan := NOT "ManAuto";
END_REGION

REGION Network 8
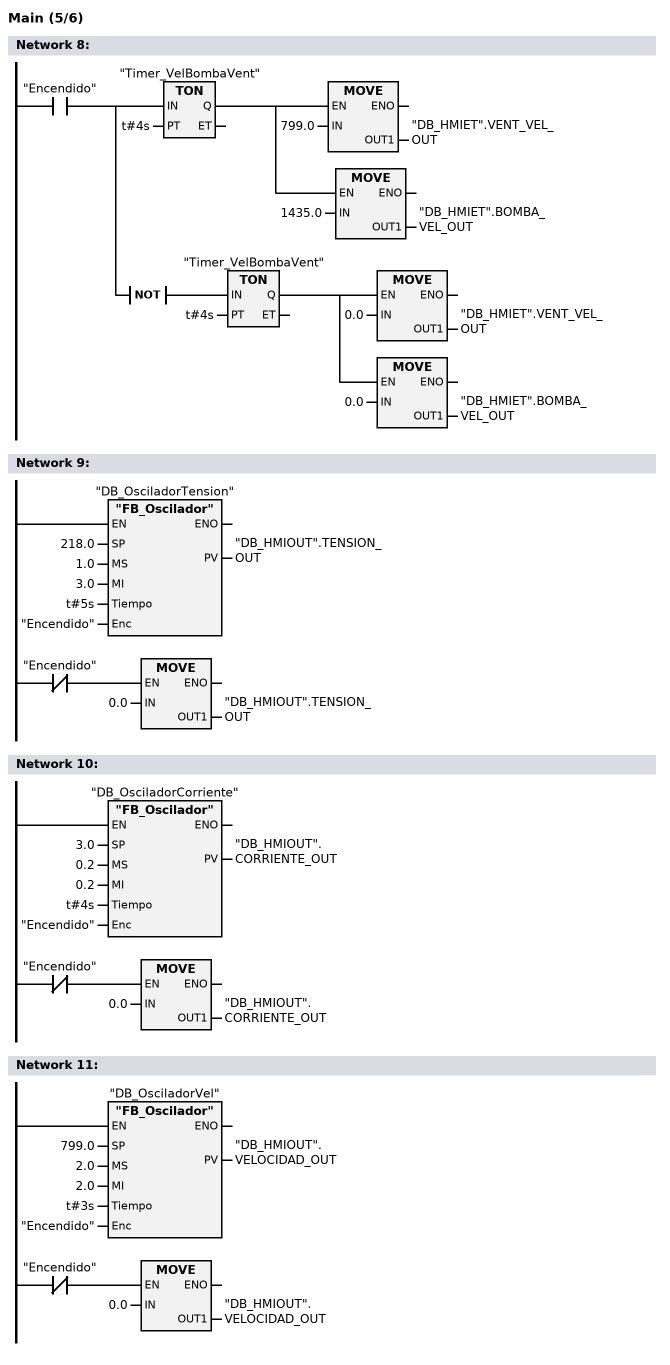
   "Timer_VelBombaVent".TON(IN := "Encendido", PT := t#4s);
   IF "Timer_VelBombaVent".Q THEN
       "DB_HMIET".VENT_VEL_OUT := 799.0;
       "DB_HMIET".BOMBA_VEL_OUT := 1435.0;
   END_IF;
   "Timer_VelBombaVent".TON(IN := NOT "Encendido", PT := t#4s);
   IF "Timer_VelBombaVent".Q THEN
       "DB_HMIET".VENT_VEL_OUT := 0.0;
       "DB_HMIET".BOMBA_VEL_OUT := 0.0;
   END_IF;
END_REGION

REGION Network 9
   RUNG wire#powerrail
      "DB_OsciladorTension"(SP := 218.0, MS := 1.0, MI := 3.0, Tiempo := t#5s, Enc := "Encendido", PV => "DB_HMIOUT".TENSION_OUT)
   END_RUNG
   RUNG wire#powerrail
      I_Contact( "Encendido" )
      Move(in := 0.0, out1 => "DB_HMIOUT".TENSION_OUT)
   END_RUNG
   // the same network as SCL:
   "DB_OsciladorTension"(SP := 218.0,   // "FB_Oscilador"
                         MS := 1.0,
                         MI := 3.0,
                         Tiempo := t#5s,
                         Enc := "Encendido",
                         PV => "DB_HMIOUT".TENSION_OUT);
   IF NOT "Encendido" THEN "DB_HMIOUT".TENSION_OUT := 0.0; END_IF;
END_REGION

REGION Network 10
   RUNG wire#powerrail
      "DB_OsciladorCorriente"(SP := 3.0, MS := 0.2, MI := 0.2, Tiempo := t#4s, Enc := "Encendido", PV => "DB_HMIOUT".CORRIENTE_OUT)
   END_RUNG
   RUNG wire#powerrail
      I_Contact( "Encendido" )
      Move(in := 0.0, out1 => "DB_HMIOUT".CORRIENTE_OUT)
   END_RUNG
   // the same network as SCL:
   "DB_OsciladorCorriente"(SP := 3.0,   // "FB_Oscilador"
                           MS := 0.2,
                           MI := 0.2,
                           Tiempo := t#4s,
                           Enc := "Encendido",
                           PV => "DB_HMIOUT".CORRIENTE_OUT);
   IF NOT "Encendido" THEN "DB_HMIOUT".CORRIENTE_OUT := 0.0; END_IF;
END_REGION

REGION Network 11
   RUNG wire#powerrail
      "DB_OsciladorVel"(SP := 799.0, MS := 2.0, MI := 2.0, Tiempo := t#3s, Enc := "Encendido", PV => "DB_HMIOUT".VELOCIDAD_OUT)
   END_RUNG
   RUNG wire#powerrail
      I_Contact( "Encendido" )
      Move(in := 0.0, out1 => "DB_HMIOUT".VELOCIDAD_OUT)
   END_RUNG
   // the same network as SCL:
   "DB_OsciladorVel"(SP := 799.0,   // "FB_Oscilador"
                     MS := 2.0,
                     MI := 2.0,
                     Tiempo := t#3s,
                     Enc := "Encendido",
                     PV => "DB_HMIOUT".VELOCIDAD_OUT);
   IF NOT "Encendido" THEN "DB_HMIOUT".VELOCIDAD_OUT := 0.0; END_IF;
END_REGION

REGION Network 12
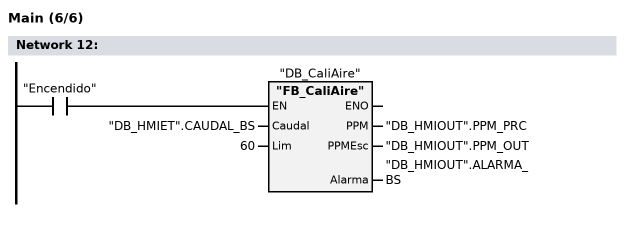
   RUNG wire#powerrail
      Contact( "Encendido" )
      "DB_CaliAire"(Caudal := "DB_HMIET".CAUDAL_BS, Lim := 60, PPM => "DB_HMIOUT".PPM_PRC, PPMEsc => "DB_HMIOUT".PPM_OUT, Alarma => "DB_HMIOUT".ALARMA_BS)
   END_RUNG
   // the same network as SCL:
   IF "Encendido" THEN
       "DB_CaliAire"(Caudal := "DB_HMIET".CAUDAL_BS,   // "FB_CaliAire"
                     Lim := 60,
                     PPM => "DB_HMIOUT".PPM_PRC,
                     PPMEsc => "DB_HMIOUT".PPM_OUT,
                     Alarma => "DB_HMIOUT".ALARMA_BS);
   END_IF;
END_REGION
END_ORGANIZATION_BLOCK